# B&R Automation Studio project POMTRS_lab_2
Automation Studio 4.2.10.53 SP

## Configuration Config1

CPU 4PP065.0571-P74, AutomationRuntime D4.52, Build 4.1.2, Vc V4.26.5

### Task classes (Cpu.sw)
```
Cyclic#1 (cycle 1000 us, tolerance 0 us):
  SimAperiod <- SimAperiodic.prg
Libraries: CtrlLib, AsIOTime
```

### Hardware
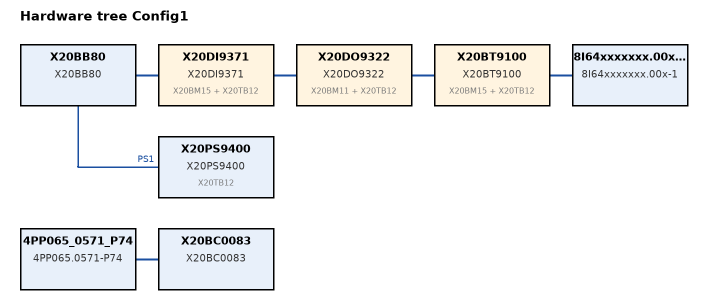
```
4PP065_0571_P74 : 4PP065.0571-P74 v1.1.1.0
  Connector IF4:
    EplInterfaceRedundant = 0
    CycleTime = 1000
    EplEthInterfaceRedundant = 0
  Connector IF5:
    ActivateDevice = 1
    Mode = Manual
    InternetAddress = 10.0.1.10
    SubnetMask = 255.255.255.0
  ConfigurationID = labBR
  TimerDeviceType = EPLX2X
  TimerDevice = 4PP065_0571_P74.IF4
  TaskClassIdleTime = 2000
  Cyclic1Duration = 1000
  Cyclic1Tolerance = 0
  Cyclic2Duration = 20000
  Cyclic2Tolerance = 20000
  Cyclic3Duration = 50000
  Cyclic3Tolerance = 50000
  Cyclic4Duration = 100000
  Cyclic4Tolerance = 100000
  Cyclic5Duration = 200000
  Cyclic5Tolerance = 200000
  Cyclic6Duration = 500000
  Cyclic6Tolerance = 500000
  Cyclic7Duration = 1000000
  Cyclic7Tolerance = 1000000
  Cyclic8Duration = 10000
  Cyclic8Tolerance = 30000000
8I64xxxxxxx.00x-1 : 8I64xxxxxxx.00x-1 v1.3.9.1  [X2X1 -> X20BT9100.X2X1]
  FunctionModel = Standard
  Supervision = off
  packedETAD = packed
  packedETI = packed
  packedCMDD = packed
  packedCMI = packed
  UNS = 220
  NCR = 10
  NSP = 890
  COS = 64
X20BB80 : X20BB80 v1.0.0.2
X20BC0083 : X20BC0083 v2.5.0.0  [PLK1 -> 4PP065_0571_P74.IF4 (NodeNumber=2); SL -> X20BB80.SL1]
X20BM11 : X20BM11 v1.0.0.1  [X2X1 -> X20BM15a.X2X2]
X20BM15 : X20BM15 v1.0.1.0  [X2X1 -> X20BM11.X2X2 (NodeNumber=10)]
X20BM15a : X20BM15 v1.0.1.0  [X2X1 -> X20BB80.IF1 (NodeNumber=5)]
X20BT9100 : X20BT9100 v1.0.2.4  [SS1 -> X20TB12a.SS; SL -> X20BM15.SL1]
X20DI9371 : X20DI9371 v1.0.1.3  [SS1 -> X20TB12b.SS; SL -> X20BM15a.SL1]
X20DO9322 : X20DO9322 v1.0.3.0  [SS1 -> X20TB12c.SS; SL -> X20BM11.SL1]
X20PS9400 : X20PS9400 v1.0.2.4  [SS1 -> X20TB12.SS; PS -> X20BB80.PS1]
X20TB12 : X20TB12 v1.0.0.0
X20TB12a : X20TB12 v1.0.0.0
X20TB12b : X20TB12 v1.0.0.0
X20TB12c : X20TB12 v1.0.0.0
```

### IoMap.iom - 4PP065_0571_P74/IoMap.iom
```iecst
VAR_CONFIG
	::GateControl.X64Ctrl.Mapping.ETAD_Input AT %IW."8I64xxxxxxx.00x-1".ETAD_Input;
	::GateControl.X64Ctrl.Mapping.CMDD_Output AT %QW."8I64xxxxxxx.00x-1".CMDD_Output;
	::GateControl.X64Ctrl.Mapping.RFRD_Input AT %IW."8I64xxxxxxx.00x-1".RFRD_Input;
	::GateControl.X64Ctrl.Mapping.LFRD_Output AT %QW."8I64xxxxxxx.00x-1".LFRD_Output;
	::GateControl.Mapping.DirectionSwitch AT %IX."X20DI9371".DigitalInput01;
	::GateControl.Mapping.SensorOpen AT %IX."X20DI9371".DigitalInput02;
	::GateControl.Mapping.SensorNearlyOpen AT %IX."X20DI9371".DigitalInput03;
	::GateControl.Mapping.SensorNearlyClose AT %IX."X20DI9371".DigitalInput04;
	::GateControl.Mapping.SensorClose AT %IX."X20DI9371".DigitalInput05;
	::GateControl.Leds.Mapping.Led1 AT %QX."X20DO9322".DigitalOutput02;
	::GateControl.Leds.Mapping.Led2 AT %QX."X20DO9322".DigitalOutput03;
	::GateControl.Leds.Mapping.Led3 AT %QX."X20DO9322".DigitalOutput04;
	::GateControl.Leds.Mapping.Led4 AT %QX."X20DO9322".DigitalOutput05;
END_VAR
```

## Logical view

Binary libraries used (declarations not repeated): operator, runtime, astime, AsIecCon, AsIOTime

### Global.var - Global variables
```iecst
VAR
	GateControl : FBGateControl;
END_VAR
```

### Package Logical/Libraries - Global libraries

### Library Logical/Libraries/CtrlLib (ANSIC)
Depends on: AsIOTime

#### Types.typ - Exported data types
```iecst
TYPE
	TX64Mapping : 	STRUCT
		RFRD_Input : INT; (*Вход RFRD*)
		LFRD_Output : INT; (*Выход LFRD*)
		CMDD_Output : UINT; (*Выход CMDD*)
		ETAD_Input : UINT; (*Вход ETAD*)
	END_STRUCT;
	TX64State :
		(
		STATE_NOT_READY_TO_SWITCH_ON := 0,
		STATE_SWITCH_ON_DISABLED := 64,
		STATE_READY_TO_SWITCH_ON := 33,
		STATE_SWITCHED_ON := 35,
		STATE_OPERATION_ENABLED := 39
		);
	TX64Command :
		(
		CMD_DISABLE_VOLTAGE := 0,
		CMD_SHUTDOWN := 6,
		CMD_SWITCH_ON := 7,
		CMD_ENABLE_OPERATION := 15
		);
	TX64Control : 	STRUCT
		Init : BOOL; (*Команда на инициализацию*)
		Enable : BOOL; (*Разрешение на работу*)
		ActSpeed : REAL; (*Актуальная скорость*)
		SetSpeed : REAL; (*Уставка по скорости*)
	END_STRUCT;
	TGateState :
		(
		ST_UNKNOWN,
		ST_OPEN,
		ST_NEARLY_OPEN,
		ST_MIDDLE,
		ST_NEARLY_CLOSED,
		ST_CLOSED
		);
	TGateLedState :
		(
		GATE_LED_BBBB,
		GATE_LED_oooo,
		GATE_LED_Oooo,
		GATE_LED_OOoo,
		GATE_LED_OOOo,
		GATE_LED_OOOO
		);
	TGatesLeds : 	STRUCT
		Led1 : BOOL;
		Led2 : BOOL;
		Led3 : BOOL;
		Led4 : BOOL;
	END_STRUCT;
	TGateMapping : 	STRUCT
		DirectionSwitch : BOOL;
		SensorOpen : BOOL;
		SensorNearlyOpen : BOOL;
		SensorNearlyClose : BOOL;
		SensorClose : BOOL;
	END_STRUCT;
END_TYPE
```

#### Constants.var - Exported constants
```iecst
VAR CONSTANT
	SPEED_HIGH : REAL := 60;
	SPEED_LOW : REAL := 6;
	SPEED_ZERO : REAL := 0.0;
END_VAR
```

#### CtrlLib.fun - Exported functions and function blocks
```iecst
FUNCTION_BLOCK FBApertiodic (*Апериодическое Звено 2-го порядка W  = 0.1 / (0.01s^2+0.3s+1). dt=0.001*) (*$GROUP=User,$CAT=User,$GROUPICON=User.png,$CATICON=User.png*)
	VAR_INPUT
		x : REAL; (*Вход*)
		init : BOOL; (*Вход инициализации*)
	END_VAR
	VAR_OUTPUT
		y : REAL; (*Выход*)
	END_VAR
	VAR
		xz2 : REAL; (*xz^-2*)
		yz2 : REAL; (*yz^-2*)
		yz1 : REAL; (*yz^-1*)
		xz1 : REAL; (*xz^-1*)
	END_VAR
END_FUNCTION_BLOCK

FUNCTION_BLOCK FBX64Ctrl (*X64 Inverter Control*) (*$GROUP=User,$CAT=User,$GROUPICON=User.png,$CATICON=User.png*)
	VAR_OUTPUT
		Control : TX64Control; (*Команды управления*)
		Mapping : TX64Mapping; (*Переменные назначаемые на частоный пробразователь*)
		State : TX64State; (*Состояние*)
	END_VAR
END_FUNCTION_BLOCK

FUNCTION_BLOCK FBGateControl (*Управление воротами*) (*$GROUP=User,$CAT=User,$GROUPICON=User.png,$CATICON=User.png*)
	VAR_INPUT
		Init : BOOL; (*Вход инициализации*)
	END_VAR
	VAR_OUTPUT
		Leds : FBGateLed;
		X64Ctrl : FBX64Ctrl; (*Функциональный блок управления частотным преобрзователем*)
		State : TGateState; (*Состояние*)
		Mapping : TGateMapping; (*Датчики и органы управления*)
	END_VAR
END_FUNCTION_BLOCK

FUNCTION_BLOCK FBGateLed (*Управление лампочками*) (*$GROUP=User,$CAT=User,$GROUPICON=User.png,$CATICON=User.png*)
	VAR_INPUT
		Init : BOOL; (*Вход инициализации*)
		LedState : TGateLedState; (*Вход уставки по состоянию лампочек*)
		StatePos : TGateState;
	END_VAR
	VAR_OUTPUT
		Mapping : TGatesLeds; (*Выходы лампочек*)
	END_VAR
	VAR
		TimestampPrev : DINT; (*Метка времени для мигания*)
		Timestamp : DINT; (*Метка времени для мигания*)
		cnt_fast : INT;
		cnt_middle : INT;
		cnt_slow : INT;
	END_VAR
END_FUNCTION_BLOCK
```

#### FBApertiodic.c
```c
#include <bur/plctypes.h>
#ifdef __cplusplus
	extern "C"
	{
#endif
	#include "CtrlLib.h"
#ifdef __cplusplus
	};
#endif
/* Апериодическое Звено 2-го порядка W  = 0.1 / (0.01s^2+0.3s+1) */
void FBApertiodic(struct FBApertiodic* inst)
{
	if(inst->init){
		inst->init = 0;
		inst->xz1=0;
		inst->xz2=0;
		inst->yz1=0;
		inst->yz2=0;
		inst->x=0;
		inst->y=0;
		return;
	}
	//Z-преобразование апериодического звена для dt=0.001 c
	inst->y=(4.9503e-06)*inst->xz1+(4.9011e-06)*inst->xz2-(-1.970347019481279)*inst->yz1-(0.9704455335485083)*inst->yz2;
	inst->xz2 = inst->xz1;
	inst->xz1 = inst->x;
	inst->yz2 = inst->yz1;
	inst->yz1 = inst->y;
}
```

#### FBX64Ctrl.c
```c
#include <bur/plctypes.h>
#ifdef __cplusplus
	extern "C"
	{
#endif
	#include "CtrlLib.h"
#ifdef __cplusplus
	};
#endif
/* X64 Inverter Control */
void FBX64Ctrl(struct FBX64Ctrl* inst)
{
	if(inst->Control.Init){
		inst->State=STATE_NOT_READY_TO_SWITCH_ON;
		inst->Control.ActSpeed=0;
		inst->Control.Enable=0;
		inst->Control.SetSpeed=0;
		inst->Mapping.CMDD_Output=0;
		inst->Mapping.LFRD_Output=0;
		inst->Mapping.ETAD_Input=0;
		inst->Mapping.RFRD_Input=0;
		inst->Control.Init=0;
		return;
	}

	inst->State=inst->Mapping.ETAD_Input & 0x006F;
	inst->Control.ActSpeed = inst->Mapping.RFRD_Input;
	inst->Control.ActSpeed = inst->Control.ActSpeed/60.0*2.0*3.1415926;

	if(!inst->Control.Enable){
		inst->Mapping.CMDD_Output = CMD_DISABLE_VOLTAGE;
		inst->Mapping.LFRD_Output=0;
	} else {
		switch(inst->State)
		{
			case STATE_NOT_READY_TO_SWITCH_ON:
				break;
			case STATE_SWITCH_ON_DISABLED:
				inst->Mapping.CMDD_Output = CMD_SHUTDOWN;
				inst->Mapping.LFRD_Output=0;
				break;
			case STATE_READY_TO_SWITCH_ON:
				inst->Mapping.CMDD_Output = CMD_SWITCH_ON;
				inst->Mapping.LFRD_Output=0;
				break;
			case STATE_SWITCHED_ON:
				inst->Mapping.CMDD_Output = CMD_ENABLE_OPERATION;
				inst->Mapping.LFRD_Output=0;
				break;
			case STATE_OPERATION_ENABLED:
				inst->Mapping.LFRD_Output=inst->Control.SetSpeed*60.0/(2.0*3.1415926);
				break;
		}
	}
}
```

#### FBGateControl.c
```c
#include <bur/plctypes.h>
#ifdef __cplusplus
	extern "C"
	{
#endif
	#include "CtrlLib.h"
#ifdef __cplusplus
	};
#endif
/* Управление воротами */
void FBGateControl(struct FBGateControl* inst)
{
	if(inst->Init){
		inst->Init = 0;
		inst->State = ST_UNKNOWN;
		inst->X64Ctrl.Control.Init = 1;
		inst->Mapping.DirectionSwitch = 0;
		inst->Mapping.SensorClose = 0;
		inst->Mapping.SensorNearlyClose = 0;
		inst->Mapping.SensorNearlyOpen = 0;
		inst->Mapping.SensorOpen = 0;
		FBX64Ctrl(&inst->X64Ctrl);
		inst->X64Ctrl.Control.Enable = 1;
		inst->Leds.Init=1;
		FBGateLed(&inst->Leds);
		return;
	}

	switch (inst->State){
		case ST_UNKNOWN:
			inst->Leds.LedState = GATE_LED_BBBB;
			if (inst->Mapping.DirectionSwitch == 0){	//Налево
				if(inst->Mapping.SensorClose){
					inst->State = ST_CLOSED;
					break;
				}
				if(inst->Mapping.SensorNearlyClose){
					inst->State = ST_NEARLY_CLOSED;
					break;
				}
				if(inst->Mapping.SensorNearlyOpen){
					inst->State = ST_MIDDLE;
					break;
				}
				if(inst->Mapping.SensorNearlyOpen){
					inst->State = ST_NEARLY_OPEN;
					break;
				}
				inst->X64Ctrl.Control.SetSpeed = -SPEED_LOW;
			} else {									//Направо
				if(inst->Mapping.SensorClose){
					inst->State = ST_NEARLY_CLOSED;
					break;
				}
				if(inst->Mapping.SensorNearlyClose){
					inst->State = ST_MIDDLE;
					break;
				}
				if(inst->Mapping.SensorNearlyOpen){
					inst->State = ST_NEARLY_OPEN;
					break;
				}
				if(inst->Mapping.SensorNearlyOpen){
					inst->State = ST_OPEN;
					break;
				}
				inst->X64Ctrl.Control.SetSpeed = SPEED_LOW;
			  }
			break;
		case ST_OPEN:
			inst->Leds.LedState = GATE_LED_oooo;
			if((inst->X64Ctrl.Control.ActSpeed>0)&&(inst->Mapping.SensorOpen==0)){
				inst->State = ST_NEARLY_OPEN;
				break;
			}
			if (inst->Mapping.DirectionSwitch == 0){	//Налево
				inst->X64Ctrl.Control.SetSpeed = -SPEED_ZERO;
			} else {									//Направо
				inst->X64Ctrl.Control.SetSpeed = SPEED_LOW;
			  }
			break;
		case ST_NEARLY_OPEN:
			inst->Leds.LedState = GATE_LED_Oooo;
			if(inst->X64Ctrl.Control.ActSpeed>0){
				if(inst->Mapping.SensorNearlyOpen){
					inst->State = ST_MIDDLE;
					break;
				}
			} else {
				if(inst->Mapping.SensorOpen){
					inst->State = ST_OPEN;
					break;
				}
              }
			if (inst->Mapping.DirectionSwitch == 0){	//Налево
				inst->X64Ctrl.Control.SetSpeed = -SPEED_LOW;
			} else {									//Направо
				inst->X64Ctrl.Control.SetSpeed = SPEED_LOW;
			  }
			break;
		case ST_MIDDLE:
			inst->Leds.LedState = GATE_LED_OOoo;
			if(inst->X64Ctrl.Control.ActSpeed>0){
				if(inst->Mapping.SensorNearlyClose){
					inst->State = ST_NEARLY_CLOSED;
					break;
				}
			} else {
				if(inst->Mapping.SensorNearlyOpen){
					inst->State = ST_NEARLY_OPEN;
					break;
				}
              }
			if (inst->Mapping.DirectionSwitch == 0){	//Налево
				inst->X64Ctrl.Control.SetSpeed = -SPEED_HIGH;
			} else {									//Направо
				inst->X64Ctrl.Control.SetSpeed = SPEED_HIGH;
			  }
			break;
		case ST_NEARLY_CLOSED:
			inst->Leds.LedState = GATE_LED_OOOo;
			if(inst->X64Ctrl.Control.ActSpeed>0){
				if(inst->Mapping.SensorClose){
					inst->State = ST_CLOSED;
					break;
				}
			} else {
				if(inst->Mapping.SensorNearlyClose){
					inst->State = ST_MIDDLE;
					break;
				}
              }
			if (inst->Mapping.DirectionSwitch == 0){	//Налево
				inst->X64Ctrl.Control.SetSpeed = -SPEED_LOW;
			} else {									//Направо
				inst->X64Ctrl.Control.SetSpeed = SPEED_LOW;
			  }
			break;
		case ST_CLOSED:
			inst->Leds.LedState = GATE_LED_OOOO;
			if((inst->X64Ctrl.Control.ActSpeed<0)&&(inst->Mapping.SensorClose==0)){
				inst->State = ST_NEARLY_CLOSED;
				break;
			}
			if (inst->Mapping.DirectionSwitch == 0){	//Налево
				inst->X64Ctrl.Control.SetSpeed = -SPEED_LOW;
			} else {									//Направо
				inst->X64Ctrl.Control.SetSpeed = SPEED_ZERO;
			  }
			break;
	}

	FBX64Ctrl(&inst->X64Ctrl);
	FBGateLed(&inst->Leds);
}
```

#### FBGateLed.c
```c
#include <bur/plctypes.h>
#ifdef __cplusplus
	extern "C"
	{
#endif
	#include "CtrlLib.h"
#ifdef __cplusplus
	};
#endif
/* Управление лампочками */
void FBGateLed(struct FBGateLed* inst)
{
	if(inst->Init){
		inst->cnt_fast = 2000;
		inst->cnt_middle = 5000;
		inst->cnt_slow = 10000;
		inst->Mapping.Led1=0;
		inst->Mapping.Led2=0;
		inst->Mapping.Led3=0;
		inst->Mapping.Led4=0;
		inst->Init=0;
		inst->LedState=GATE_LED_BBBB;
		inst->Timestamp = AsIOTimeCyclicStart();;
		inst->TimestampPrev = inst->Timestamp;
		return;
	}

	inst->Timestamp = AsIOTimeCyclicStart();

	switch (inst->LedState){
		case GATE_LED_BBBB:
				if((inst->Timestamp-inst->TimestampPrev)>=500000){
					inst->Mapping.Led1=!inst->Mapping.Led1;
					inst->TimestampPrev=inst->Timestamp;
				}
				inst->Mapping.Led2=inst->Mapping.Led1;
				inst->Mapping.Led3=inst->Mapping.Led1;
				inst->Mapping.Led4=inst->Mapping.Led1;
			break;
		case GATE_LED_oooo:
			inst->Mapping.Led1=0;
			inst->Mapping.Led2=0;
			inst->Mapping.Led3=0;
			inst->Mapping.Led4=0;
			break;
		case GATE_LED_Oooo:
			if(inst->StatePos = ST_NEARLY_OPEN)
			{
				inst->cnt_slow = inst->cnt_slow - 1;
				if(inst->cnt_slow == 0)
				{
					inst->Mapping.Led1 = !inst->Mapping.Led1;
					inst->cnt_slow = 1000;
				}
			}
			inst->Mapping.Led2=0;
			inst->Mapping.Led3=0;
			inst->Mapping.Led4=0;
			break;
		case GATE_LED_OOoo:
			if(inst->StatePos = ST_MIDDLE)
			{
				inst->cnt_fast = inst->cnt_fast - 1;
				if(inst->cnt_fast == 0)
				{
					inst->Mapping.Led1=!inst->Mapping.Led1;
					inst->Mapping.Led2=!inst->Mapping.Led2;
					inst->cnt_fast = 100;
				}
			}
			inst->Mapping.Led3=0;
			inst->Mapping.Led4=0;
			break;
		case GATE_LED_OOOo:
			if(inst->StatePos = ST_NEARLY_CLOSED)
			{
				inst->cnt_slow = inst->cnt_slow - 1;
				if(inst->cnt_slow == 0)
				{
					inst->Mapping.Led1=!inst->Mapping.Led1;
					inst->Mapping.Led2=!inst->Mapping.Led2;
					inst->Mapping.Led3=!inst->Mapping.Led3;
					inst->cnt_slow = 1000;
				}
			}
			inst->Mapping.Led4=0;
			break;

		case GATE_LED_OOOO:
			inst->Mapping.Led1=0;
			inst->Mapping.Led2=0;
			inst->Mapping.Led3=0;
			inst->Mapping.Led4=0;
			break;
	}
}
```

### Program Logical/SimAperiodic (ANSIC)

#### Main.c
```c
#include <bur/plctypes.h>

#ifdef _DEFAULT_INCLUDES
	#include <AsDefault.h>
#endif

void _INIT ProgramInit(void)
{
	GateControl.Init=1;
	FBGateControl(&GateControl);
}

void _CYCLIC ProgramCyclic(void)
{
	FBGateControl(&GateControl);
}

void _EXIT ProgramExit(void)
{

}
```

Listed in the project but not available here: Logical/Global.typ
